// TIA Portal V20 export
VAR_GLOBAL   // PLC tag table "Sonplas_Inputs"
   DI_SonplasDiagDPCoupler AT %I200.0 : Bool;
   DI_SonplasReady AT %I200.1 : Bool;
   DI_SonplasNoEStop AT %I200.2 : Bool;
   DI_SonplasDoorsClosed AT %I200.3 : Bool;
   DI_SonplasRunError AT %I200.4 : Bool;
   DI_SonplasFreeI200_5 AT %I200.5 : Bool;
   DI_SonplasFreeI200_6 AT %I200.6 : Bool;
   DI_SonplasFreeI200_7 AT %I200.7 : Bool;
   DI_SonplasFreeI201_0 AT %I201.0 : Bool;
   DI_SonplasOutCollision AT %I201.1 : Bool;
   DI_SonplasFreeI201_2 AT %I201.2 : Bool;
   DI_SonplasFreeI201_3 AT %I201.3 : Bool;
   DI_SonplasFreeI201_4 AT %I201.4 : Bool;
   DI_SonplasFreeI201_5 AT %I201.5 : Bool;
   DI_SonplasFreeI201_6 AT %I201.6 : Bool;
   DI_SonplasFreeI201_7 AT %I201.7 : Bool;
   DI_SonplasShuttle1Finished AT %I202.0 : Bool;
   DI_SonplasFreeI202_1 AT %I202.1 : Bool;
   DI_SonplasFreeI202_2 AT %I202.2 : Bool;
   DI_SonplasFreeI202_3 AT %I202.3 : Bool;
   DI_SonplasFreeI202_4 AT %I202.4 : Bool;
   DI_SonplasFreeI202_5 AT %I202.5 : Bool;
   DI_SonplasFreeI202_6 AT %I202.6 : Bool;
   DI_SonplasFreeI202_7 AT %I202.7 : Bool;
   DI_SonplasShuttle2Finished AT %I203.0 : Bool;
   DI_SonplasFreeI203_1 AT %I203.1 : Bool;
   DI_SonplasFreeI203_2 AT %I203.2 : Bool;
   DI_SonplasFreeI203_3 AT %I203.3 : Bool;
   DI_SonplasFreeI203_4 AT %I203.4 : Bool;
   DI_SonplasFreeI203_5 AT %I203.5 : Bool;
   DI_SonplasFreeI203_6 AT %I203.6 : Bool;
   DI_SonplasFreeI203_7 AT %I203.7 : Bool;
   DI_SonplasFlowResultAvail AT %I244.0 : Bool;
   DI_SonplasFreeI244_1 AT %I244.1 : Bool;
   DI_SonplasFreeI244_2 AT %I244.2 : Bool;
   DI_SonplasFreeI244_3 AT %I244.3 : Bool;
   DI_SonplasFreeI244_4 AT %I244.4 : Bool;
   DI_SonplasFreeI244_5 AT %I244.5 : Bool;
   DI_SonplasFreeI244_6 AT %I244.6 : Bool;
   DI_SonplasFreeI244_7 AT %I244.7 : Bool;
   AI_SonplasDMC_Code1 AT %IB204 : Byte;
   AI_SonplasDMC_Code2 AT %IB224 : Byte;
   AI_SonplasFlowResult AT %IW245 : Word;
   AI_SonplasDMC_CodeFlow AT %IB247 : Byte;
END_VAR
